PROGRAM main
VAR
	Enable AT %QX0.0 : bool;
	Output AT %QX0.1 : bool;
END_VAR

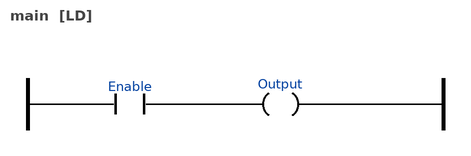
(* LD diagram, written out as Structured Text *)
Output := Enable;
END_PROGRAM
